FUNCTION_BLOCK TcoTier EXTENDS TcoCore.TcoObject
VAR
	_nextExpectedCycle : ULINT;
END_VAR

{attribute 'hide'}
METHOD FB_init : BOOL
VAR_INPUT
	bInitRetains : BOOL; // if TRUE, the retain variables are initialized (warm start / cold start)
	bInCopyCode : BOOL;  // if TRUE, the instance afterwards gets moved into the copy code (online change)
	ParentObject : ITcoObject;	
END_VAR
END_METHOD

METHOD IsNewTier : BOOL
IsNewTier := THIS^.Context.StartCycleCount <> _nextExpectedCycle;
_nextExpectedCycle := THIS^.Context.StartCycleCount + 1;
END_METHOD

END_FUNCTION_BLOCK

(* stored: Version 1.1.0.1, ProductVersion 3.1.4024.9
   POU TcoTier: Id {b03c48ad-ab45-0697-3bbf-4f1922cef1af}, SpecialFunc None
   Method FB_init: Id {ff9e5ffa-34d3-0196-37e7-07844c34c44c}
   Method IsNewTier: Id {f55c3d87-5b7f-04ae-3379-eb9ac260e42d} *)
